% RSLogix 500 project P4_BAK022.RSS, saved by version 12.00.00.00 %
PROJECT "UNTITLED"    % processor: Bul.1763 MicroLogix 1100 Series B %

PROGRAM FILES
  LAD 2 "MAIN"  4 rungs
  LAD 3 "DIGITAL IO"  7 rungs
  LAD 4 "CONTROLS"  15 rungs
  LAD 5 "STATUS"  6 rungs

DATA FILES
  O0 OUTPUT  4 elements
  I1 INPUT  6 elements
  S2 STATUS  66 elements
  B3 BINARY  2 elements
  T4 TIMER  3 elements
  C5 COUNTER  1 elements
  R6 CONTROL  1 elements
  N7 INTEGER  1 elements
  F8 FLOAT  1 elements

LADDER 2 "MAIN"
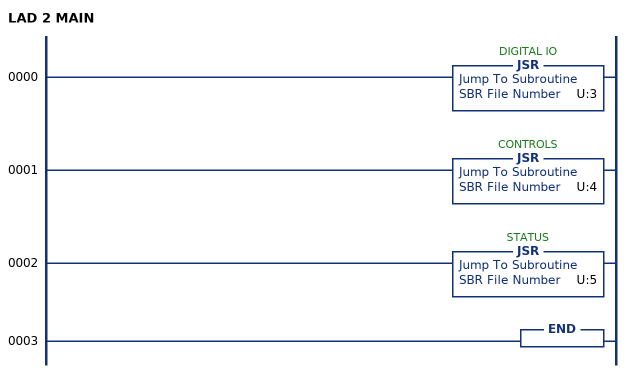
% Rung: 0 %
SOR JSR U:3 EOR
%   U:3  "DIGITAL IO" %
% Rung: 1 %
SOR JSR U:4 EOR
%   U:4  "CONTROLS" %
% Rung: 2 %
SOR JSR U:5 EOR
%   U:5  "STATUS" %
% Rung: 3 %
SOR END EOR

LADDER 3 "DIGITAL IO"
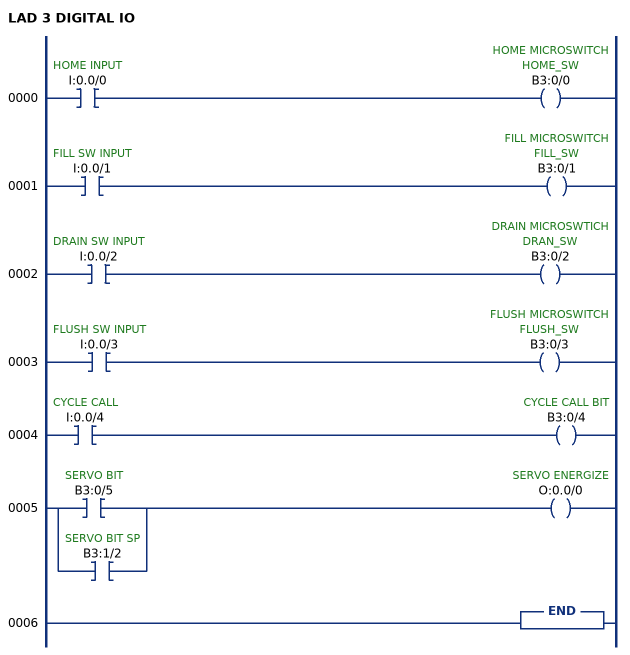
% Rung: 0 %
SOR XIC I:0.0/0 OTE B3:0/0 EOR
%   I:0.0/0  "HOME INPUT" %
%   B3:0/0  HOME_SW  "HOME MICROSWITCH" %
% Rung: 1 %
SOR XIC I:0.0/1 OTE B3:0/1 EOR
%   I:0.0/1  "FILL SW INPUT" %
%   B3:0/1  FILL_SW  "FILL MICROSWITCH" %
% Rung: 2 %
SOR XIC I:0.0/2 OTE B3:0/2 EOR
%   I:0.0/2  "DRAIN SW INPUT" %
%   B3:0/2  DRAN_SW  "DRAIN MICROSWTICH" %
% Rung: 3 %
SOR XIC I:0.0/3 OTE B3:0/3 EOR
%   I:0.0/3  "FLUSH SW INPUT" %
%   B3:0/3  FLUSH_SW  "FLUSH MICROSWITCH" %
% Rung: 4 %
SOR XIC I:0.0/4 OTE B3:0/4 EOR
%   I:0.0/4  "CYCLE CALL" %
%   B3:0/4  "CYCLE CALL BIT" %
% Rung: 5 %
SOR BST XIC B3:0/5 NXB XIC B3:1/2 BND OTE O:0.0/0 EOR
%   B3:0/5  "SERVO BIT" %
%   B3:1/2  "SERVO BIT SP" %
%   O:0.0/0  "SERVO ENERGIZE" %
% Rung: 6 %
SOR END EOR

LADDER 4 "CONTROLS"
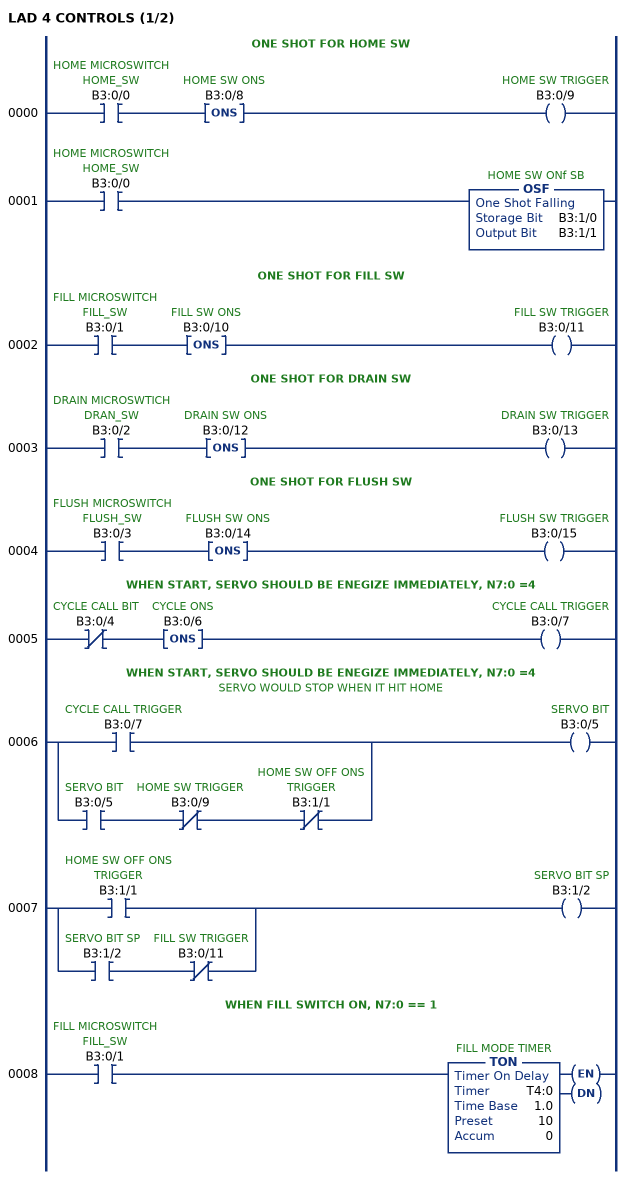
% Rung: 0 %
% TITLE: ONE SHOT FOR HOME SW %
SOR XIC B3:0/0 ONS B3:0/8 OTE B3:0/9 EOR
%   B3:0/0  HOME_SW  "HOME MICROSWITCH" %
%   B3:0/8  "HOME SW ONS" %
%   B3:0/9  "HOME SW TRIGGER" %
% Rung: 1 %
SOR XIC B3:0/0 OSF B3:1/0 B3:1/1 EOR
%   B3:0/0  HOME_SW  "HOME MICROSWITCH" %
%   B3:1/0  "HOME SW ONf SB" %
%   B3:1/1  "HOME SW OFF ONS TRIGGER" %
% Rung: 2 %
% TITLE: ONE SHOT FOR FILL SW %
SOR XIC B3:0/1 ONS B3:0/10 OTE B3:0/11 EOR
%   B3:0/1  FILL_SW  "FILL MICROSWITCH" %
%   B3:0/10  "FILL SW ONS" %
%   B3:0/11  "FILL SW TRIGGER" %
% Rung: 3 %
% TITLE: ONE SHOT FOR DRAIN SW %
SOR XIC B3:0/2 ONS B3:0/12 OTE B3:0/13 EOR
%   B3:0/2  DRAN_SW  "DRAIN MICROSWTICH" %
%   B3:0/12  "DRAIN SW ONS" %
%   B3:0/13  "DRAIN SW TRIGGER" %
% Rung: 4 %
% TITLE: ONE SHOT FOR FLUSH SW %
SOR XIC B3:0/3 ONS B3:0/14 OTE B3:0/15 EOR
%   B3:0/3  FLUSH_SW  "FLUSH MICROSWITCH" %
%   B3:0/14  "FLUSH SW ONS" %
%   B3:0/15  "FLUSH SW TRIGGER" %
% Rung: 5 %
% TITLE: WHEN START, SERVO SHOULD BE ENEGIZE IMMEDIATELY, N7:0 =4 %
SOR XIO B3:0/4 ONS B3:0/6 OTE B3:0/7 EOR
%   B3:0/4  "CYCLE CALL BIT" %
%   B3:0/6  "CYCLE ONS" %
%   B3:0/7  "CYCLE CALL TRIGGER" %
% Rung: 6 %
% TITLE: WHEN START, SERVO SHOULD BE ENEGIZE IMMEDIATELY, N7:0 =4 %
% SERVO WOULD STOP WHEN IT HIT HOME %
SOR BST XIC B3:0/7 NXB XIC B3:0/5 XIO B3:0/9 XIO B3:1/1 BND OTE B3:0/5 EOR
%   B3:0/7  "CYCLE CALL TRIGGER" %
%   B3:0/5  "SERVO BIT" %
%   B3:0/9  "HOME SW TRIGGER" %
%   B3:1/1  "HOME SW OFF ONS TRIGGER" %
% Rung: 7 %
SOR BST XIC B3:1/1 NXB XIC B3:1/2 XIO B3:0/11 BND OTE B3:1/2 EOR
%   B3:1/1  "HOME SW OFF ONS TRIGGER" %
%   B3:1/2  "SERVO BIT SP" %
%   B3:0/11  "FILL SW TRIGGER" %
% Rung: 8 %
% TITLE: WHEN FILL SWITCH ON, N7:0 == 1 %
SOR XIC B3:0/1 TON T4:0 1.0 10 0 EOR
%   B3:0/1  FILL_SW  "FILL MICROSWITCH" %
%   T4:0  "FILL MODE TIMER" %

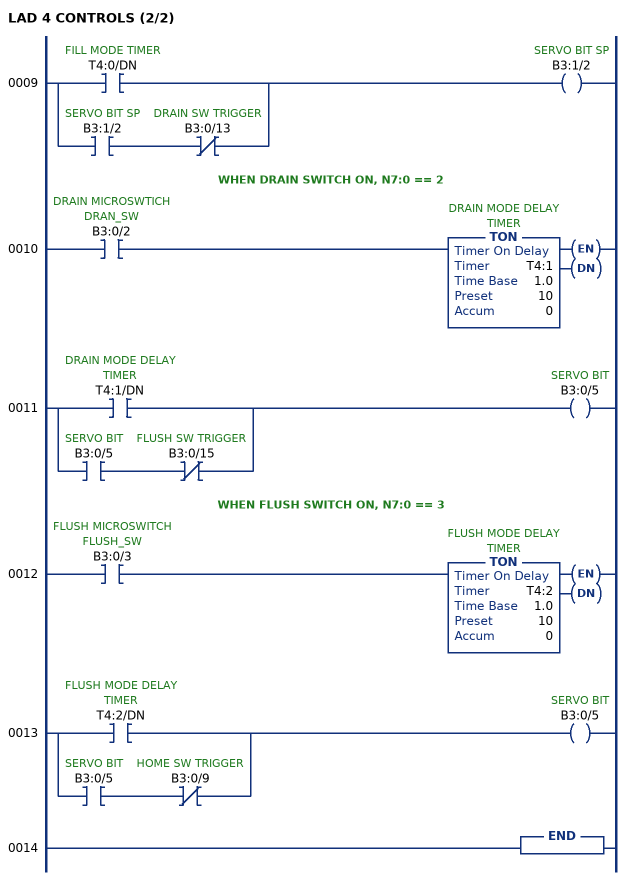
% Rung: 9 %
SOR BST XIC T4:0/DN NXB XIC B3:1/2 XIO B3:0/13 BND OTE B3:1/2 EOR
%   T4:0  "FILL MODE TIMER" %
%   B3:1/2  "SERVO BIT SP" %
%   B3:0/13  "DRAIN SW TRIGGER" %
% Rung: 10 %
% TITLE: WHEN DRAIN SWITCH ON, N7:0 == 2 %
SOR XIC B3:0/2 TON T4:1 1.0 10 0 EOR
%   B3:0/2  DRAN_SW  "DRAIN MICROSWTICH" %
%   T4:1  "DRAIN MODE DELAY TIMER" %
% Rung: 11 %
SOR BST XIC T4:1/DN NXB XIC B3:0/5 XIO B3:0/15 BND OTE B3:0/5 EOR
%   T4:1  "DRAIN MODE DELAY TIMER" %
%   B3:0/5  "SERVO BIT" %
%   B3:0/15  "FLUSH SW TRIGGER" %
% Rung: 12 %
% TITLE: WHEN FLUSH SWITCH ON, N7:0 == 3 %
SOR XIC B3:0/3 TON T4:2 1.0 10 0 EOR
%   B3:0/3  FLUSH_SW  "FLUSH MICROSWITCH" %
%   T4:2  "FLUSH MODE DELAY TIMER" %
% Rung: 13 %
SOR BST XIC T4:2/DN NXB XIC B3:0/5 XIO B3:0/9 BND OTE B3:0/5 EOR
%   T4:2  "FLUSH MODE DELAY TIMER" %
%   B3:0/5  "SERVO BIT" %
%   B3:0/9  "HOME SW TRIGGER" %
% Rung: 14 %
SOR END EOR

LADDER 5 "STATUS"
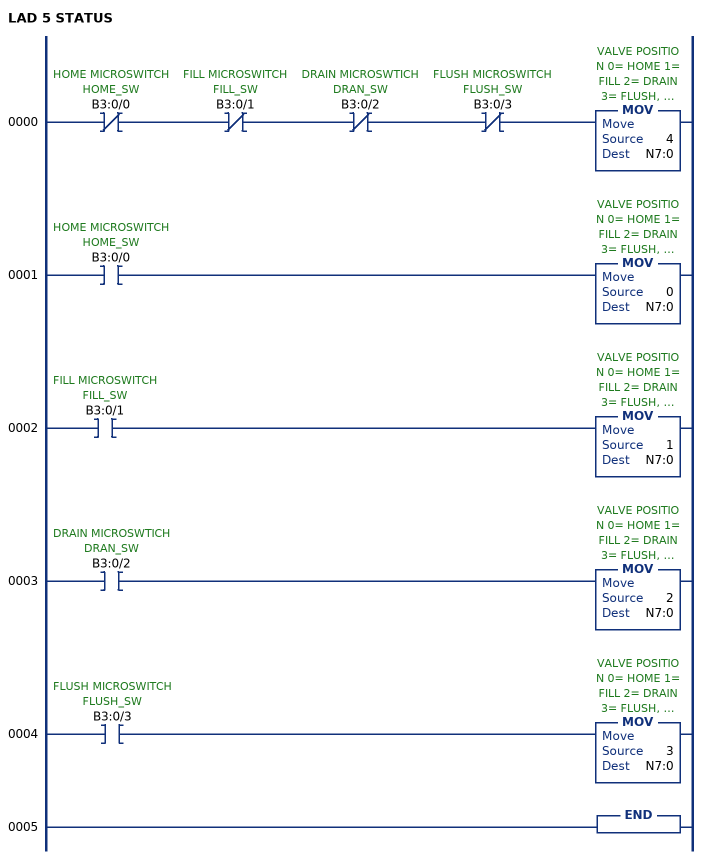
% Rung: 0 %
SOR XIO B3:0/0 XIO B3:0/1 XIO B3:0/2 XIO B3:0/3 MOV 4 N7:0 EOR
%   B3:0/0  HOME_SW  "HOME MICROSWITCH" %
%   B3:0/1  FILL_SW  "FILL MICROSWITCH" %
%   B3:0/2  DRAN_SW  "DRAIN MICROSWTICH" %
%   B3:0/3  FLUSH_SW  "FLUSH MICROSWITCH" %
%   N7:0  "VALVE POSITION 0= HOME 1= FILL 2= DRAIN 3= FLUSH, 4 TRAVELLI" %
% Rung: 1 %
SOR XIC B3:0/0 MOV 0 N7:0 EOR
%   B3:0/0  HOME_SW  "HOME MICROSWITCH" %
%   N7:0  "VALVE POSITION 0= HOME 1= FILL 2= DRAIN 3= FLUSH, 4 TRAVELLI" %
% Rung: 2 %
SOR XIC B3:0/1 MOV 1 N7:0 EOR
%   B3:0/1  FILL_SW  "FILL MICROSWITCH" %
%   N7:0  "VALVE POSITION 0= HOME 1= FILL 2= DRAIN 3= FLUSH, 4 TRAVELLI" %
% Rung: 3 %
SOR XIC B3:0/2 MOV 2 N7:0 EOR
%   B3:0/2  DRAN_SW  "DRAIN MICROSWTICH" %
%   N7:0  "VALVE POSITION 0= HOME 1= FILL 2= DRAIN 3= FLUSH, 4 TRAVELLI" %
% Rung: 4 %
SOR XIC B3:0/3 MOV 3 N7:0 EOR
%   B3:0/3  FLUSH_SW  "FLUSH MICROSWITCH" %
%   N7:0  "VALVE POSITION 0= HOME 1= FILL 2= DRAIN 3= FLUSH, 4 TRAVELLI" %
% Rung: 5 %
SOR END EOR

DATA TABLE (non-zero values as saved)
DATA T4
% .PRE .ACC %
% T4:0 % 10 0
% T4:1 % 10 0
% T4:2 % 10 0
